% RSLogix 500 project Controlador_implementado.RSS, saved by version 8.30.00.16 %
PROJECT "P4131222"    % processor: Bul.1763 MicroLogix 1100 Series B %

PROGRAM FILES
  LAD 2   14 rungs

DATA FILES
  O0 OUTPUT  6 elements
  I1 INPUT  12 elements
  S2 STATUS  66 elements
  B3 BINARY  1 elements
  T4 TIMER  1 elements
  C5 COUNTER  1 elements
  R6 CONTROL  1 elements
  N7 INTEGER  10 elements
  F8 FLOAT  9 elements
  PD9   1 elements

LADDER 2
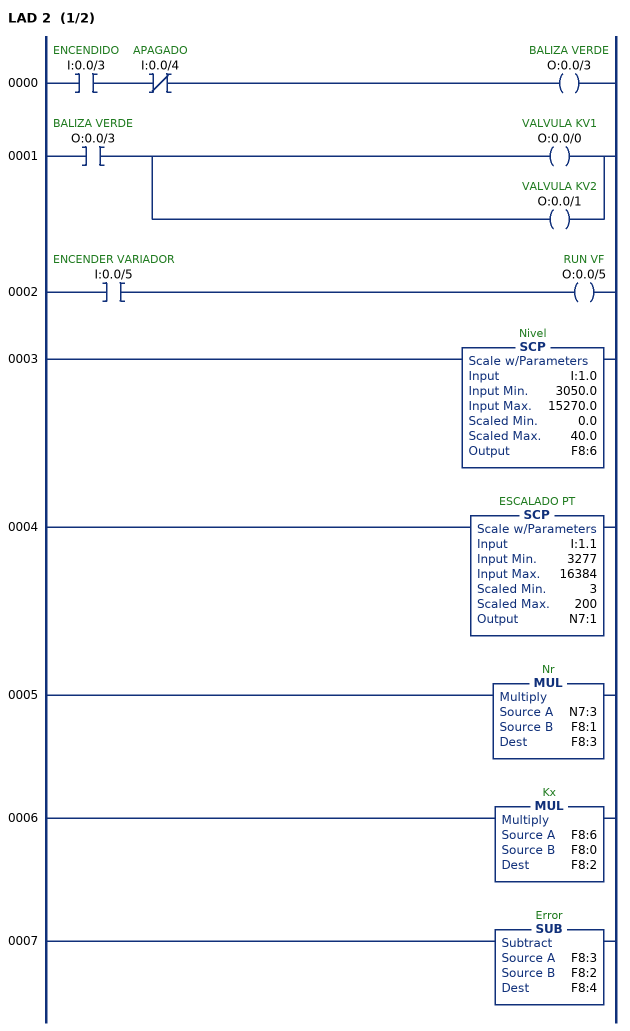
% Rung: 0 %
SOR XIC I:0.0/3 XIO I:0.0/4 OTE O:0.0/3 EOR
%   I:0.0/3  "ENCENDIDO" %
%   I:0.0/4  "APAGADO" %
%   O:0.0/3  "BALIZA VERDE" %
% Rung: 1 %
SOR XIC O:0.0/3 BST OTE O:0.0/0 NXB OTE O:0.0/1 BND EOR
%   O:0.0/3  "BALIZA VERDE" %
%   O:0.0/0  "VALVULA KV1" %
%   O:0.0/1  "VALVULA KV2" %
% Rung: 2 %
SOR XIC I:0.0/5 OTE O:0.0/5 EOR
%   I:0.0/5  "ENCENDER VARIADOR" %
%   O:0.0/5  "RUN VF" %
% Rung: 3 %
SOR SCP I:1.0 3050.0 15270.0 0.0 40.0 F8:6 EOR
%   I:1.0  "LT" %
%   F8:6  "Nivel" %
% Rung: 4 %
SOR SCP I:1.1 3277 16384 3 200 N7:1 EOR
%   I:1.1  "PT" %
%   N7:1  "ESCALADO PT" %
% Rung: 5 %
SOR MUL N7:3 F8:1 F8:3 EOR
%   N7:3  "SET POINT" %
%   F8:1  "N" %
%   F8:3  "Nr" %
% Rung: 6 %
SOR MUL F8:6 F8:0 F8:2 EOR
%   F8:6  "Nivel" %
%   F8:0  "K" %
%   F8:2  "Kx" %
% Rung: 7 %
SOR SUB F8:3 F8:2 F8:4 EOR
%   F8:3  "Nr" %
%   F8:2  "Kx" %
%   F8:4  "Error" %

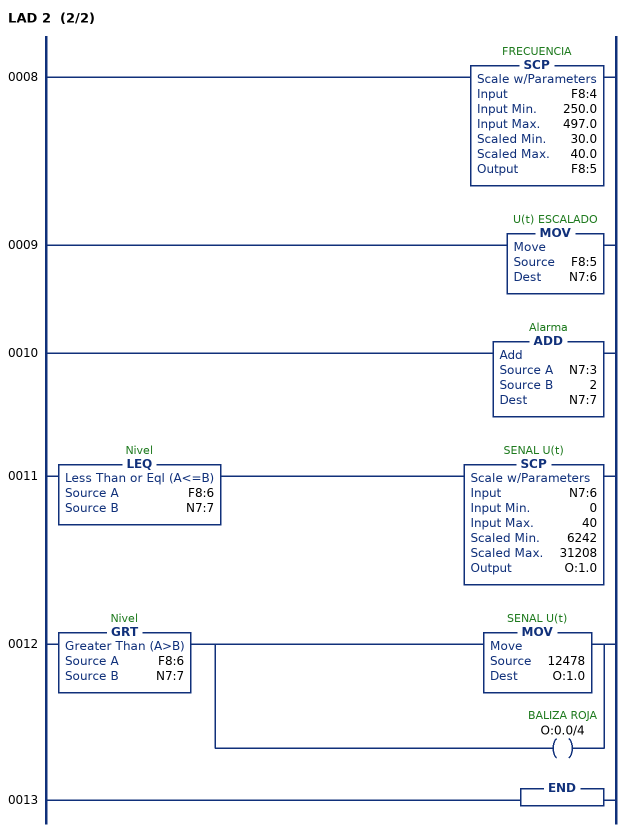
% Rung: 8 %
SOR SCP F8:4 250.0 497.0 30.0 40.0 F8:5 EOR
%   F8:4  "Error" %
%   F8:5  "FRECUENCIA" %
% Rung: 9 %
SOR MOV F8:5 N7:6 EOR
%   F8:5  "FRECUENCIA" %
%   N7:6  "U(t) ESCALADO" %
% Rung: 10 %
SOR ADD N7:3 2 N7:7 EOR
%   N7:3  "SET POINT" %
%   N7:7  "Alarma" %
% Rung: 11 %
SOR LEQ F8:6 N7:7 SCP N7:6 0 40 6242 31208 O:1.0 EOR
%   F8:6  "Nivel" %
%   N7:7  "Alarma" %
%   N7:6  "U(t) ESCALADO" %
%   O:1.0  "SENAL U(t)" %
% Rung: 12 %
SOR GRT F8:6 N7:7 BST MOV 12478 O:1.0 NXB OTE O:0.0/4 BND EOR
%   F8:6  "Nivel" %
%   N7:7  "Alarma" %
%   O:1.0  "SENAL U(t)" %
%   O:0.0/4  "BALIZA ROJA" %
% Rung: 13 %
SOR END EOR

OTHER DOCUMENTED ADDRESSES
  B3:0/0  "STOP"
  N7:0  "ESCALADO LT"
  N7:2  "ERROR"
  N7:4  "Nr(t)"
  N7:5  "Kx(t)"
  N7:9  F8
  PD9:0.2  "REFERENCIA"
  PD9:0.3  "Kc"
  PD9:0.4  "Ti"
  PD9:0.5  "Td"

DATA TABLE (non-zero values as saved)
DATA N7
% N7:0 % 0 1 0 20 0 0 27 22 -6 10
DATA F8
% F8:0 % 2.6499 8.8889 0.8153539 177.778 176.9626
% F8:5 % 27.04302 0.3076923 0 0
